// TIA Portal V16 export
// export: Created 2024-08-30T11:36:05.1698106Z, ExportSetting WithDefaults, DisplayName Totally Integrated Automation Portal, DisplayVersion V16, DisplayName TIA Portal Version Control Interface, DisplayVersion V16, DisplayName TIA Portal Openness, DisplayVersion V16, DisplayName STEP 7 Professional, DisplayVersion V16, DisplayName STEP 7 Safety, DisplayVersion V16, DisplayName WinCC Professional, DisplayVersion V16
DATA_BLOCK "DB00852_St_ConstAqScaleData"   // DB852
TITLE = Static DB [SYSTEM CONSTANTS] — Analog Input Scale Data and Ranges
{ S7_Optimized_Access := 'TRUE' }
AUTHOR : M_Gledhill
FAMILY : SysConstants
NAME : St_ConstAiScaleData
VERSION : 1.0
// PRACTICAL SERIES AUTOMATION LIBRARY (PAL)   —   COPYRIGHT 2020 – M. GLEDHILL (MIT LICENCE)
//                   ———— ◆ ————
// FULL ONLINE DOCUMENTATION IS AVAILABLE AT: https://practicalseries.com/2001-pal/index.html
// stored: AutoNumber false, DBAccessibleFromOPCUA true, IsOnlyStoredInLoadMemory false, IsRetainMemResEnabled false, IsWriteProtectedInAS false, MemoryReserve 100
   VAR
      _DB_Header { ExternalAccessible := 'False'; ExternalVisible := 'False'; ExternalWritable := 'False'} : Array[0..79] of Bool;   // Static DB [SYSTEM CONSTANTS] — Analog Instrument Scale Data and Ranges
      __________0000_0 { ExternalAccessible := 'False'; ExternalVisible := 'False'; ExternalWritable := 'False'} : Bool := false;
      __________0000_1 { ExternalAccessible := 'False'; ExternalVisible := 'False'; ExternalWritable := 'False'} : Bool := false;
      revInfo { ExternalWritable := 'False'} : "UT01000_St_SysRevision";
      __________0010_0 { ExternalAccessible := 'False'; ExternalVisible := 'False'; ExternalWritable := 'False'} : Bool := false;
      __________0010_1 { ExternalAccessible := 'False'; ExternalVisible := 'False'; ExternalWritable := 'False'} : Bool := false;   // ▀▀▀▀ ANALOG SCALE SIGNALS — MODULATING VALVES
      AQ_SCALE_FCV001_DMD { ExternalWritable := 'False'; S7_SetPoint := 'True'} : "UT00852_Sy_ConstAqScaleData";   // Inlet flow control valve position demand (0 to 100%)
      __________0020_0 { ExternalAccessible := 'False'; ExternalVisible := 'False'; ExternalWritable := 'False'} : Bool := false;
      __________0020_1 { ExternalAccessible := 'False'; ExternalVisible := 'False'; ExternalWritable := 'False'} : Bool := false;   // ▀▀▀▀ ANALOG SCALE SIGNALS — CHART RECORDER
      AQ_SCALE_REC001 { ExternalWritable := 'False'; S7_SetPoint := 'True'} : "UT00852_Sy_ConstAqScaleData";   // Recorder - Inlet flow meter (0-100 l/s)
      AQ_SCALE_REC002 { ExternalWritable := 'False'; S7_SetPoint := 'True'} : "UT00852_Sy_ConstAqScaleData";   // Recorder - Inlet tank level (0-50 m3)
   END_VAR
BEGIN
   // _DB_Header[0] : ▄▄▄▄▄▄▄▄▄▄▄▄▄▄▄▄▄▄▄▄▄▄▄▄▄▄▄▄▄▄▄▄ ＣＯＮＳＴＡＮＴＳ ▄▄
   // _DB_Header[2] : TITLE: SYSTEM CONSTANTS — ANALOG INPUT SCALE DATA AND RANGES
   // _DB_Header[4] : ▀▀▀▀▀▀▀▀▀▀▀▀▀▀▀▀▀▀▀▀▀▀▀▀▀▀▀▀▀▀▀▀▀▀▀▀▀▀▀▀▀▀▀▀
   // _DB_Header[5] : TYPE: STATIC
   // _DB_Header[6] : ▄▄▄▄▄▄▄▄▄▄▄▄▄▄▄▄▄▄▄▄▄▄▄▄▄▄▄▄▄▄▄▄▄▄▄▄▄▄▄▄ ʷᴵᴰ⁻ᵈʰᵇ ▄
   // _DB_Header[8] : DB00852_St_ConstAqScaleData is a static data block that holds a full set of scaled ranges,
   // _DB_Header[9] : engineering units, device tag and descriptive data for all types of analog output scaled signals.
   // _DB_Header[11] : Each dataset is stored in a structure of user data type: UT00852_St_ConstAqScaleData.
   // _DB_Header[12] : This structure is configured to hold all the data required to name, scale and apply engineering
   // _DB_Header[13] : units to an analog output signal.
   // _DB_Header[15] : All the scaled signal data is stored as constants and is used by all modules that have an interface
   // _DB_Header[16] : to an analog output card.
   // _DB_Header[18] : The purpose of the user data type and associated data block is to provide a consistent set of
   // _DB_Header[19] : scaled ranges and other data for each device that is available to the Controller
   // _DB_Header[20] : as an analog output.
   // _DB_Header[22] : The ranges correspond to the scaled values of a signal that is to be converted into an analog
   // _DB_Header[23] : output, for example, a modulating valve may have a scaled range of 0% to 100%.
   // _DB_Header[25] : In addition, each dataset contains the device tag (e.g. FCV001), the engineering
   // _DB_Header[26] : units in use (e.g. l/s, kg/hour, °C, % &c.), over-range and under-range limits, a textual description
   // _DB_Header[27] : of the function of the device e.g.inlet flow control valve and additional user specific
   // _DB_Header[28] : information.
   // _DB_Header[30] : The PDF version of the SMDS for this module is available online here:
   // _DB_Header[31] : http://psop.uk/pal-smds-db00851-p
   // _DB_Header[33] : ━━━ ⬙⬙⬙⬙⬙⬙ ━━━
   // _DB_Header[35] : ▄▄▄▄▄▄▄▄▄▄▄▄▄▄▄▄▄▄▄▄▄▄▄▄▄▄▄▄▄▄▄▄▄▄▄▄▄▄▄▄▄▄▄▄
   // _DB_Header[36] : MODIFICATION HISTORY
   // _DB_Header[38] : This is a summary of the recent software modifications made to this block (most recent at top)
   // _DB_Header[40] : ―――――――――――――――――――――――――――――――――――――――――――
   // _DB_Header[41] : DATE REVISION MASTER BRANCH DEV
   // _DB_Header[42] : (nnn.amm) COMMIT TAG (Base ---> Merge) BRANCH Author
   // _DB_Header[43] : ———————————————————————————————————————————
   // _DB_Header[44] : 2024.05.17 001.000 D0017A-000.104 D0017 N/A D0017A M. Gledhill
   // _DB_Header[45] : DB00852 — RELEASED FOR USE
   // _DB_Header[47] : 2024.05.03 000.801 D0017A-000.102 D0017 N/A D0017A M. Gledhill
   // _DB_Header[48] : DB00852 Block populated
   // _DB_Header[50] : 2024.04.09 000.101 D0017A-000.101 D0017 N/A D0017A M. Gledhill
   // _DB_Header[51] : DB00852 Block created
   // _DB_Header[52] : ———————————————————————————————————————————
   // _DB_Header[53] : Where: nnn = Major revision
   // _DB_Header[54] : a = Type (1-7 Development, 8 Proving, 9 Qualification, 0 Release)
   // _DB_Header[55] : mm = Minor revision (must be 00 if a = 0)
   // _DB_Header[56] : Block properties version number should be set to nn.a (only one decimal place)
   // _DB_Header[58] : ██████████████ █ █ █ █ END █ █ █ █ ██████████████
   revInfo.REV_BLOCK := 'DB00852';
   revInfo.REV_NUMBER := '001.000';
   revInfo.REV_DATE := '2024-05-17';
   revInfo.REV_AUTHOR := 'M. Gledhill';
   AQ_SCALE_FCV001_DMD.AQ_TAG := 'FCV001';
   AQ_SCALE_FCV001_DMD.SCALE_MIN := 0.0;
   AQ_SCALE_FCV001_DMD.SCALE_MAX := 100.0;
   AQ_SCALE_FCV001_DMD.SCALE_UNITS := '%';
   AQ_SCALE_FCV001_DMD.SCALE_DESC := 'Inlet flow control valve (0 to 100%)';
   AQ_SCALE_FCV001_DMD.LIMIT_UNDER := -2.5;
   AQ_SCALE_FCV001_DMD.LIMIT_OVER := 102.5;
   AQ_SCALE_FCV001_DMD.USER_INFO_1 := 'Instrument manufacturer: Siemens';
   AQ_SCALE_FCV001_DMD.USER_INFO_2 := 'Instrument type: 2-port magnetic';
   AQ_SCALE_FCV001_DMD.USER_INFO_3 := 'Instrument part no.: MXG461.15-0.6';
   AQ_SCALE_FCV001_DMD.USER_INFO_4 := 'Instrument serial no.:2075181118';
   AQ_SCALE_REC001.AQ_TAG := 'REC001';
   AQ_SCALE_REC001.SCALE_MIN := 0.0;
   AQ_SCALE_REC001.SCALE_MAX := 100.0;
   AQ_SCALE_REC001.SCALE_UNITS := 'l/s';
   AQ_SCALE_REC001.SCALE_DESC := 'Recorder - Inlet flow meter (0-100 l/s)';
   AQ_SCALE_REC002.AQ_TAG := 'REC002';
   AQ_SCALE_REC002.SCALE_MIN := 0.0;
   AQ_SCALE_REC002.SCALE_MAX := 50.0;
   AQ_SCALE_REC002.SCALE_UNITS := 'm3';
   AQ_SCALE_REC002.SCALE_DESC := 'Recorder - Inlet tank level (0-50 m3)';
END_DATA_BLOCK
